// Mitsubishi GX Works2 project: GT_EX1   PLC: Q03UDV

PROGRAM MAIN
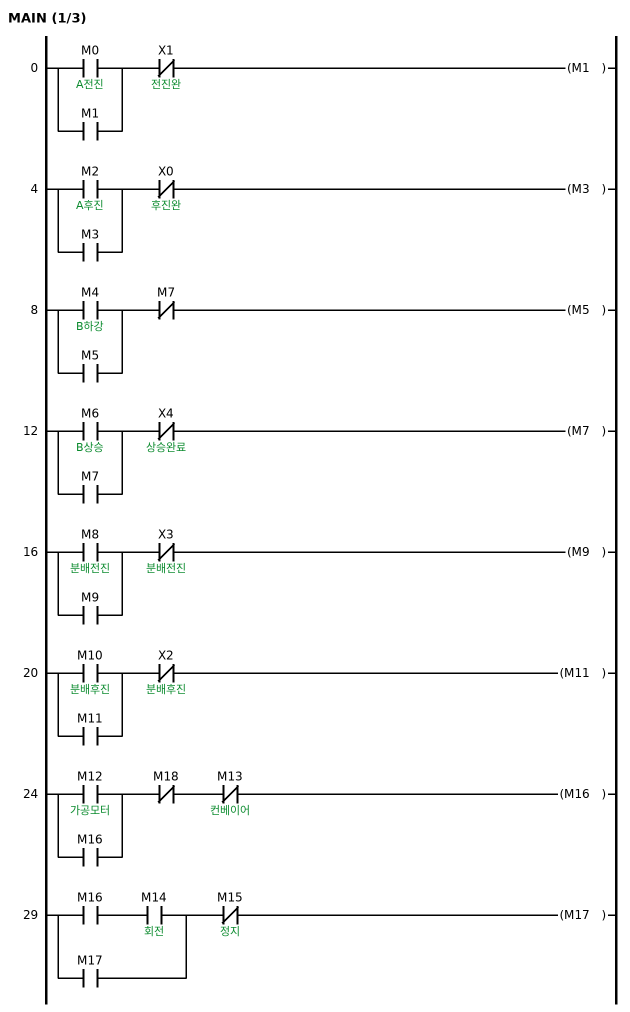
0     LD      M0  ; A전진
      OR      M1
      ANI     X1  ; 전진완
      OUT     M1
4     LD      M2  ; A후진
      OR      M3
      ANI     X0  ; 후진완
      OUT     M3
8     LD      M4  ; B하강
      OR      M5
      ANI     M7
      OUT     M5
12    LD      M6  ; B상승
      OR      M7
      ANI     X4  ; 상승완료
      OUT     M7
16    LD      M8  ; 분배전진
      OR      M9
      ANI     X3  ; 분배전진
      OUT     M9
20    LD      M10  ; 분배후진
      OR      M11
      ANI     X2  ; 분배후진
      OUT     M11
24    LD      M12  ; 가공모터
      OR      M16
      ANI     M18
      ANI     M13  ; 컨베이어
      OUT     M16
29    LD      M16
      AND     M14  ; 회전
      OR      M17
      ANI     M15  ; 정지
      OUT     M17
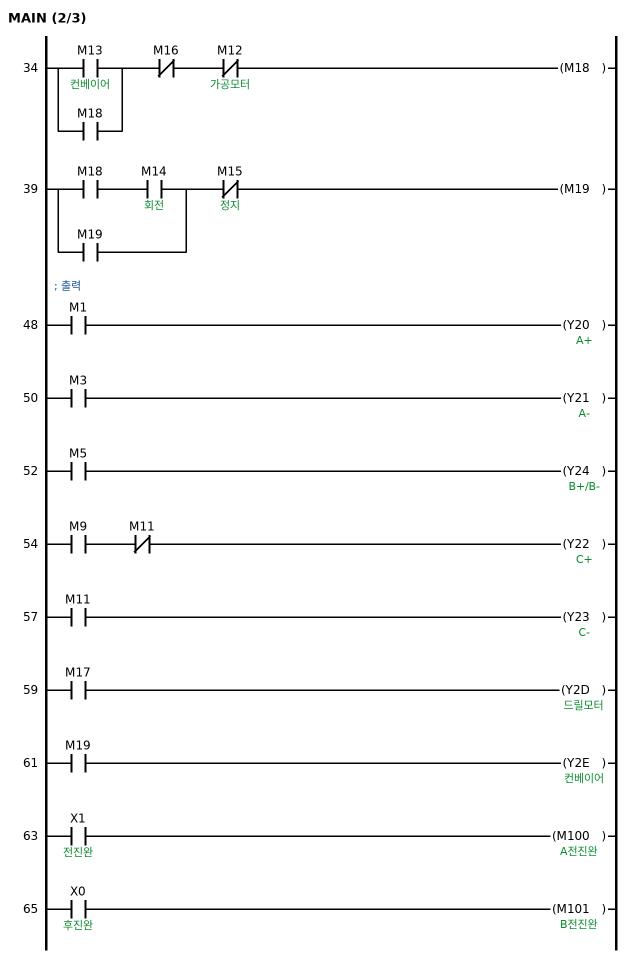
34    LD      M13  ; 컨베이어
      OR      M18
      ANI     M16
      ANI     M12  ; 가공모터
      OUT     M18
39    LD      M18
      AND     M14  ; 회전
      OR      M19
      ANI     M15  ; 정지
      OUT     M19
; 출력
48    LD      M1
      OUT     Y20  ; A+
50    LD      M3
      OUT     Y21  ; A-
52    LD      M5
      OUT     Y24  ; B+/B-
54    LD      M9
      ANI     M11
      OUT     Y22  ; C+
57    LD      M11
      OUT     Y23  ; C-
59    LD      M17
      OUT     Y2D  ; 드릴모터
61    LD      M19
      OUT     Y2E  ; 컨베이어
63    LD      X1  ; 전진완
      OUT     M100  ; A전진완
65    LD      X0  ; 후진완
      OUT     M101  ; B전진완
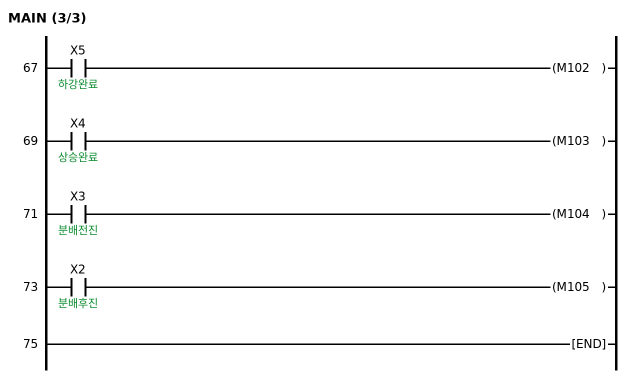
67    LD      X5  ; 하강완료
      OUT     M102
69    LD      X4  ; 상승완료
      OUT     M103
71    LD      X3  ; 분배전진
      OUT     M104
73    LD      X2  ; 분배후진
      OUT     M105
75    END
END_PROGRAM
